(*
SPDX-FileCopyrightText: © 2026 Oleksandr Tiutyk <trofimich@gmail.com>
SPDX-License-Identifier: MIT
License: https://opensource.org/license/mit
*)

(*!
<summary>Reports an argument value outside the range accepted by the caller.</summary>
<description>
The caller determines that the argument is invalid; Throw formats the diagnostic rather than validating the
argument. Argument values are represented in at most 255 characters. STRING and WSTRING values longer than 255
characters retain their first 254 characters followed by an ellipsis. Dynamic exceptions belong to the current
task memory manager until cleanup. Dynamic copies are explicitly registered by Clone after construction; plain
__NEW does not transfer ownership to the task manager.
</description>
*)

{attribute 'enable_dynamic_creation'}
{attribute 'no_explicit_call' := 'do not call this function block directly'}
FUNCTION_BLOCK ArgumentOutOfRangeException EXTENDS GeneralException IMPLEMENTS IArgumentOutOfRangeException
VAR_STAT
	//! <summary>Class name shared by all instances of this function block.</summary>
	{attribute 'hide'} 
	_ClassName : STRING := __POUNAME();
END_VAR

{attribute 'monitoring' := 'call'}
PROPERTY ClassName : REFERENCE TO STRING
GET
ClassName REF= _ClassName;
END_GET
END_PROPERTY

(*!
<summary>Creates a task-owned copy of this exception and its diagnostic payload.</summary>
<description>
Registers the newly constructed instance before copying payload, outside FB_init. Registration failure
releases the unregistered instance and raises a terminal error; copy failure leaves the registered instance
owned by the task manager for cleanup. Custom overrides must follow the same ownership sequence. The returned
reference is borrowed until task cleanup and must not be deleted by the caller.
</description>
*)
METHOD Clone : IObject
VAR
	exceptionClone : POINTER TO ArgumentOutOfRangeException;
END_VAR
exceptionClone := __NEW(ArgumentOutOfRangeException);

IF exceptionClone = 0 THEN
	DynamicMemoryManager.RaiseAllocationFailure();
END_IF

DynamicMemoryManager.RegisterAutoDisposedObject(autoDisposedObject := exceptionClone^);

exceptionClone^.CopyGeneralFields(sourceException := THIS^);

Clone := exceptionClone^;
END_METHOD

(*!
<summary>Provides the library namespace used in diagnostics.</summary>
<description>
Borrowed read-only reference to the compiler-initialized library namespace; no ownership transfer.
</description>
*)
{attribute 'monitoring' := 'call'}
PROPERTY NamespaceName : REFERENCE TO STRING
GET
NamespaceName REF= CurrentNamespace.Name;
END_GET
END_PROPERTY

(*!
<summary>Reports the byte size of this concrete instance.</summary>
<description>
Uses XSIZEOF on the instance. Does not include separately allocated payloads or prove that an arbitrary
address is valid.
</description>
*)
{attribute 'monitoring' := 'call'}
PROPERTY SelfSize : ULINT
GET
SelfSize := XSIZEOF(THIS^);
END_GET
END_PROPERTY

(*!
<summary>Formats the rejected argument and propagates the exception with source metadata.</summary>
<description>
Call in the owning cyclic task, not during FB_init. Reads the supplied value only during this call and retains
its formatted text without heap allocation during message preparation. Long STRING and WSTRING values use a
254-character prefix followed by an ellipsis; exactly 255 characters are kept unchanged. Other types use the
shared ANY formatter. Sets error code to zero and has no inner cause. Exception clone allocation failure uses
the terminal memory mechanism.
</description>
<param name="argumentName">Name of the argument rejected by the caller.</param>
<param name="argumentValue">Live value to describe; string inputs must be null-terminated.</param>
*)
METHOD Throw
VAR_INPUT
	sourceNamespaceName : STRING;
	sourceClassName : STRING;
	sourcePOUName : STRING;
	sourcePosition : STRING;
	argumentName : STRING;
	argumentValue : ANY;
END_VAR
VAR
	valueAsString : WSTRING(255);
	message : ERROR_MESSAGE;
END_VAR
valueAsString := WideStrings.AnyToStringFit255(value := argumentValue);

WideStrings.Append255(
	message,
	"Argument '",
	TO_WSTRING(argumentName),
	"' has invalid value '",
	valueAsString,
	"' in '",
	TO_WSTRING(GetFullPOUName(
		sourceNamespaceName := sourceNamespaceName,
		sourceClassName := sourceClassName,
		sourcePOUName := sourcePOUName
	)),
	"'");

InternalThrow(
	sourceNamespaceName := sourceNamespaceName,
	sourceClassName := sourceClassName,
	sourcePOUName := sourcePOUName,
	sourcePosition := sourcePosition,
	message := message,
	errorCode := 0,
	innerException := 0
);
END_METHOD

END_FUNCTION_BLOCK

(* stored: Version 1.1.0.1
   POU ArgumentOutOfRangeException: Id {98d20286-f8bd-41e5-8b87-fcb4b5d7ca5e}, SpecialFunc None
   Property ClassName: Id {c27874b7-4abc-48c2-950c-b0bb5f01f34d}
   Get Get: Id {731dacbe-6b4c-4a54-a726-b999af608436}
   Method Clone: Id {cce15318-1da6-4dd9-8b2e-884a82dd488e}
   Property NamespaceName: Id {905b7564-223e-4161-86fe-e47bcc939f12}
   Get Get: Id {d388c6b1-588b-4ade-aeba-27a186862023}
   Property SelfSize: Id {527aeda2-b68e-4925-b9c4-ca5bfdb83414}
   Get Get: Id {8dbf744f-7964-4344-9744-8dc5f4e021dd}
   Method Throw: Id {5feec76b-4654-49c9-b2bc-8cf052990d28} *)
